screen "滑块角度" 800x480
   Circle "圆_2" at 245,51 size 21x21
      Appearance <- "360"
   Circle "圆_3" at 274,56 size 21x21
      Appearance <- "10度"
   Circle "圆_4" at 303,66 size 21x21
      Appearance <- "20度"
   Circle "圆_5" at 326,79 size 21x21
      Appearance <- "30度"
   Circle "圆_6" at 346,95 size 21x21
      Appearance <- "40度"
   Circle "圆_7" at 364,115 size 21x21
      Appearance <- "50"
   Circle "圆_8" at 377,135 size 21x21
      Appearance <- "60"
   Circle "圆_9" at 385,157 size 21x21
      Appearance <- "70"
   Circle "圆_10" at 392,179 size 21x21
      Appearance <- "80"
   Circle "圆_11" at 394,202 size 21x21
      Appearance <- "90"
   Circle "圆_12" at 391,226 size 21x21
      Appearance <- "100"
   Circle "圆_13" at 386,249 size 21x21
      Appearance <- "110"
   Circle "圆_14" at 378,271 size 21x21
      Appearance <- "120"
   Circle "圆_15" at 365,292 size 21x21
      Appearance <- "130"
   Circle "圆_16" at 348,311 size 21x21
      Appearance <- "140"
   Circle "圆_17" at 328,328 size 21x21
      Appearance <- "150"
   Circle "圆_18" at 306,342 size 21x21
      Appearance <- "160"
   Circle "圆_19" at 276,353 size 21x21
      Appearance <- "170"
   Circle "圆_20" at 247,357 size 21x21
      Appearance <- "180"
   Circle "圆_22" at 219,352 size 21x21
      Appearance <- "190"
   Circle "圆_23" at 195,344 size 21x21
      Appearance <- "200"
   Circle "圆_24" at 172,333 size 21x21
      Appearance <- "210"
   Circle "圆_25" at 152,319 size 21x21
      Appearance <- "220"
   Circle "圆_26" at 133,302 size 21x21
      Appearance <- "230"
   Circle "圆_27" at 117,281 size 21x21
      Appearance <- "240"
   Circle "圆_28" at 104,258 size 21x21
      Appearance <- "250"
   Circle "圆_29" at 96,229 size 21x21
      Appearance <- "260"
   Circle "圆_30" at 93,201 size 21x21
      Appearance <- "270"
   Circle "圆_32" at 95,178 size 21x21
      Appearance <- "280"
   Circle "圆_33" at 100,155 size 21x21
      Appearance <- "290"
   Circle "圆_34" at 110,131 size 21x21
      Appearance <- "300"
   Circle "圆_35" at 126,111 size 21x21
      Appearance <- "310"
   Circle "圆_36" at 144,91 size 21x21
      Appearance <- "320"
   Circle "圆_37" at 167,74 size 21x21
      Appearance <- "330"
   Circle "圆_38" at 191,63 size 21x21
      Appearance <- "340"
   Circle "圆_39" at 218,54 size 21x21
      Appearance <- "350"
   TextField "文本域_2" at 422,193 size 43x40; Text '90'
   TextField "文本域_3" at 221,378 size 62x40; Text '180'
   TextField "文本域_5" at 196,174 size 117x31; Text '滑块位置'
   TextField "文本域_9" at 467,193 size 93x25; Text '当前产量'
   TextField "文本域_4" at 25,203 size 62x40; Text '270'
   TextField "文本域_1" at 241,12 size 24x40; Text '0'
   SymbolLibrary "符号库_1" at 405,7 size 109x71
   SymbolLibrary "符号库_2" at 646,29 size 86x40
   TextField "文本域_7" at 637,83 size 77x21; Text '滑块电机'
   TextField "文本域_6" at 423,85 size 59x21; Text '主电机'
   TextField "文本域_8" at 467,127 size 93x25; Text '设置产量'
   TextField "文本域_10" at 693,127 size 93x25; Text '计数清零'
   TextField "文本域_13" at 586,126 size 93x25; Text '计数通断'
   TextField "文本域_11" at 35,338 size 93x25; Text '润滑检测'
   TextField "文本域_12" at 454,341 size 85x23; Text '润滑故障'
   TextField "文本域_15" at 583,14 size 33x17; Text '向上'
   TextField "文本域_16" at 738,15 size 33x17; Text '向下'
   Button "按钮_1" at 28,424 size 67x56; TextOff '滑块角度'
      on Click: ActivateScreen("滑块角度", 0)
   Button "按钮_2" at 96,424 size 67x56; TextOff '设备状态'
      on Click: ActivateScreen("设备状态", 0)
   Button "按钮_3" at 163,424 size 71x55; TextOff '工作台操作'
      on Click: ActivateScreen("工作台操作", 0)
   Button "按钮_4" at 235,424 size 69x56; TextOff '气垫操作'
      on Click: ActivateScreen("气垫操作", 0)
   Button "按钮_5" at 304,423 size 66x57; TextOff '故障显示'
      on Click: ActivateScreen("故障显示", 0)
   Button "按钮_6" at 371,423 size 73x57; TextOff '输出显示'
      on Click: ActivateScreen("输出显示", 0)
   Button "按钮_7" at 445,422 size 66x58; TextOff '输入显示'
      on Click: ActivateScreen("输入显示", 0)
   IOField "I/O 域_1" at 228,215 size 56x32; FormatPattern 999
      ProcessValue <- "横梁编码器 _DB_0.11"
   IOField "I/O 域_2" at 478,153 size 81x29; FormatPattern 9999
      ProcessValue <- "ECamdata _DB_设置产量"
   Button "按钮_8" at 514,423 size 68x56; TextOn '滑块调整'; TextOff '滑块调整'
      on Click: ActivateScreen("滑块调整", 0)
   Button "按钮_9" at 667,421 size 65x58; TextOff '报警信息'
      on Click: ActivateScreen("报警信息", 0)
   Button "按钮_10" at 585,423 size 77x55; TextOff '行程控制'
      on Click: ActivateScreen("行程控制", 0)
   Circle "圆_1" at 436,26 size 35x35
      Appearance <- "主电机正转运行"
   Circle "圆_21" at 584,33 size 33x33
      Appearance <- "滑块调整向上"
   Circle "圆_31" at 738,34 size 33x33
      Appearance <- "滑块调整向下"
   IOField "I/O 域_3" at 478,219 size 87x32; FormatPattern 9999
      ProcessValue <- "IEC_Counter_0_DB_4_CV"
   Rectangle "矩形_1" at 479,258 size 88x60
      Appearance <- "产量到达"
   TextField "文本域_14" at 478,277 size 85x23; Text '产量完成'
   Switch "开关_1" at 579,170 size 102x93; CaptionText 'Switch'; TextOff '断'; TextOn '通'
      ProcessValue <- "计数开始"
      Appearance <- "计数开始"
   Button "按钮_11" at 702,187 size 75x72; TextOff '清零'
      on Press: SetBit("计数清零")
      on Release: ResetBit("计数清零")
   Circle "圆_42" at 23,374 size 35x35
      Appearance <- "横梁1分油器检测"
   Circle "圆_43" at 129,375 size 35x35
      Appearance <- "平衡器分油器检测"
   Circle "圆_44" at 481,373 size 35x35
      Appearance <- "润滑正常"
   Circle "圆_45" at 230,100 size 55x55
      Appearance <- "上死点"
   TextField "文本域_17" at 233,118 size 47x17; Text '上死点'
   Circle "圆_46" at 229,274 size 55x55
      Appearance <- "下死点"
   TextField "文本域_18" at 232,292 size 47x17; Text '下死点'
   TextField "文本域_19" at 621,339 size 85x23; Text '平衡气压'
   Circle "圆_47" at 657,374 size 35x35
      Appearance <- "平衡缸气压检测"
   TextField "文本域_20" at 705,339 size 85x23; Text '液压保护'
   Circle "圆_48" at 737,373 size 35x35
      Appearance <- "液压保护故障(1)"
   TextField "文本域_21" at 539,340 size 85x23; Text '离制压力'
   Circle "圆_49" at 568,372 size 35x35
      Appearance <- "离制压力正常"
   TextField "文本域_22" at 370,342 size 85x23; Text '急停故障'
   Circle "圆_50" at 405,372 size 35x35
      Appearance <- "安全正常(1)"
   Circle "圆_51" at 78,375 size 35x35
      Appearance <- "滑块分油器检测"
   TextField "文本域_23" at 24,385 size 33x17; Text '横梁'
   TextField "文本域_24" at 78,385 size 33x17; Text '滑块'
   TextField "文本域_25" at 124,385 size 47x17; Text '平衡缸'
   Button "按钮_12" at 740,434 size 56x44; TextOff '润滑状态'
      on Click: ActivateScreen("润滑状态", 0)

screen "设备状态" 800x480
   TextField "文本域_1" at 63,79 size 101x27; Text '润滑正常'
   TextField "文本域_2" at 64,142 size 101x27; Text '急停正常'
   TextField "文本域_3" at 50,205 size 125x27; Text '工作台夹紧'
   TextField "文本域_4" at 66,268 size 101x27; Text '气压正常'
   TextField "文本域_5" at 46,331 size 149x27; Text '液压保护正常'
   Circle "圆_1" at 325,208 size 27x27
      Appearance <- "工作台落到位前"
   TextField "文本域_6" at 293,237 size 96x16; Text '工作台前落到为'
   Circle "圆_2" at 427,207 size 27x27
      Appearance <- "工作台落到位后"
   TextField "文本域_7" at 395,237 size 96x16; Text '工作台后落到为'
   TextField "文本域_8" at 495,237 size 96x16; Text '工作台夹紧压力'
   Circle "圆_4" at 223,207 size 27x27
      Appearance <- "工作台夹紧阀(1)"
   TextField "文本域_9" at 198,237 size 83x16; Text '工作台夹紧阀'
   Circle "圆_5" at 427,81 size 27x27
      Appearance <- "润滑油压正常"
   TextField "文本域_10" at 399,111 size 83x16; Text '润滑油压正常'
   TextField "文本域_12" at 295,111 size 96x16; Text '润滑过滤器正常'
   Circle "圆_8" at 222,81 size 27x27
      Appearance <- "工作台落到位后"
   TextField "文本域_13" at 196,111 size 83x16; Text '润滑油位正常'
   Circle "圆_9" at 527,81 size 27x27
      Appearance <- "工作台落到位后"
   TextField "文本域_14" at 502,111 size 83x16; Text '润滑频次正常'
   Circle "圆_10" at 325,270 size 27x27
      Appearance <- "工作台落到位前"
   TextField "文本域_15" at 306,299 size 70x16; Text '离合器压力'
   Circle "圆_11" at 427,269 size 27x27
      Appearance <- "工作台落到位后"
   Circle "圆_12" at 223,269 size 27x27
      Appearance <- "平衡缸气压检测"
   TextField "文本域_16" at 200,298 size 70x16; Text '平衡缸压力'
   TextField "文本域_17" at 407,300 size 70x16; Text '制动器压力'
   Circle "圆_6" at 615,81 size 27x27
      Appearance <- "润滑油泵启动OK"
   TextField "文本域_11" at 590,111 size 83x16; Text '润滑电机启动'
   TextField "文本域_19" at 312,171 size 57x16; Text '急停闭点'
   TextField "文本域_20" at 207,171 size 57x16; Text '急停开点'
   TextField "文本域_21" at 414,171 size 57x16; Text '梯子开关'
   TextField "文本域_23" at 306,362 size 70x16; Text '卸荷阀卸荷'
   Circle "圆_19" at 427,332 size 27x27
      Appearance <- "液压保护故障"
   TextField "文本域_24" at 200,361 size 83x16; Text '液压保护压力'
   TextField "文本域_25" at 407,363 size 57x16; Text '系统压力'
   Button "按钮_1" at 28,424 size 67x56; TextOn '滑块角度'; TextOff '滑块角度'
      on Click: ActivateScreen("滑块角度", 0)
   Button "按钮_2" at 96,424 size 67x56; TextOn '设备状态'; TextOff '设备状态'
      on Click: ActivateScreen("设备状态", 0)
   Button "按钮_3" at 163,424 size 71x55; TextOn '工作台操作'; TextOff '工作台操作'
      on Click: ActivateScreen("工作台操作", 0)
   Button "按钮_4" at 235,424 size 69x56; TextOn '气垫操作'; TextOff '气垫操作'
      on Click: ActivateScreen("气垫操作", 0)
   Button "按钮_5" at 304,423 size 66x57; TextOn '故障显示'; TextOff '故障显示'
      on Click: ActivateScreen("故障显示", 0)
   Button "按钮_6" at 371,423 size 73x57; TextOn '输出显示'; TextOff '输出显示'
      on Click: ActivateScreen("输出显示", 0)
   Button "按钮_7" at 445,422 size 66x58; TextOn '输入显示'; TextOff '输入显示'
      on Click: ActivateScreen("输入显示", 0)
   Button "按钮_8" at 514,423 size 68x56; TextOn '滑块调整'; TextOff '滑块调整'
      on Click: ActivateScreen("滑块调整", 0)
   Button "按钮_9" at 592,422 size 65x58; TextOn '报警信息'; TextOff '报警信息'
      on Click: ActivateScreen("报警信息", 0)

screen "输入显示" 800x480
   Button "按钮_1" at 28,424 size 67x56; TextOn '滑块角度'; TextOff '滑块角度'
      on Click: ActivateScreen("滑块角度", 0)
   Button "按钮_2" at 96,424 size 67x56; TextOn '设备状态'; TextOff '设备状态'
      on Click: ActivateScreen("设备状态", 0)
   Button "按钮_3" at 163,424 size 71x55; TextOn '工作台操作'; TextOff '工作台操作'
      on Click: ActivateScreen("工作台操作", 0)
   Button "按钮_4" at 235,424 size 69x56; TextOn '气垫操作'; TextOff '气垫操作'
      on Click: ActivateScreen("气垫操作", 0)
   Button "按钮_5" at 304,423 size 66x57; TextOn '故障显示'; TextOff '故障显示'
      on Click: ActivateScreen("故障显示", 0)
   Button "按钮_6" at 371,423 size 73x57; TextOn '输出显示'; TextOff '输出显示'
      on Click: ActivateScreen("输出显示", 0)
   Button "按钮_7" at 445,422 size 66x58; TextOn '输入显示'; TextOff '输入显示'
      on Click: ActivateScreen("输入显示", 0)
   Button "按钮_8" at 514,423 size 68x56; TextOn '滑块调整'; TextOff '滑块调整'
      on Click: ActivateScreen("滑块调整", 0)
   Button "按钮_9" at 592,422 size 65x58; TextOn '报警信息'; TextOff '报警信息'
      on Click: ActivateScreen("报警信息", 0)
   TextField "文本域_1" at 10,10 size 112x19; Text '主电机零速'
      Appearance <- "主电机零速"
   TextField "文本域_2" at 10,40 size 117x19; Text '主电机温度检测'
      Appearance <- "主电机温度检测(1)"
   TextField "文本域_3" at 10,70 size 117x19; Text '调速装置正常'
      Appearance <- "主电机调速装置正常"
   TextField "文本域_4" at 10,100 size 117x19; Text '主电机风扇空开'
      Appearance <- "主电机风扇空开"
   TextField "文本域_5" at 10,130 size 117x19; Text '风扇流量检测'
      Appearance <- "主电机风扇流量检测(1)"
   TextField "文本域_8" at 10,220 size 112x19; Text '按钮站插入'
      Appearance <- "按钮站插入"
   TextField "文本域_9" at 10,250 size 112x19; Text '右前急停按钮'
      Appearance <- "右前急停按钮"
   TextField "文本域_10" at 10,280 size 112x19; Text '左前急停按钮'
      Appearance <- "左前急停按钮"
   TextField "文本域_11" at 10,310 size 112x19; Text '右后急停按钮'
      Appearance <- "右后急停按钮"
   TextField "文本域_12" at 10,340 size 112x19; Text '左后急停按钮'
      Appearance <- "左后急停按钮"
   TextField "文本域_13" at 10,370 size 112x19; Text '前安全栓'
      Appearance <- "前安全栓"
   TextField "文本域_14" at 10,400 size 112x19; Text '后安全栓'
      Appearance <- "后安全栓"
   TextField "文本域_15" at 150,220 size 119x19; Text '气垫调整空开'
      Appearance <- "气垫调整空开"
   TextField "文本域_16" at 150,250 size 119x19; Text '气垫调整上极限'
      Appearance <- "气垫调整上极限"
   TextField "文本域_17" at 150,280 size 119x19; Text '气垫调整上极限'
      Appearance <- "气垫调整下极限"
   TextField "文本域_18" at 150,310 size 119x19; Text '冷却电机过热'
      Appearance <- "气垫冷却电机过热"
   TextField "文本域_19" at 150,340 size 119x19; Text '气垫左落下到位'
      Appearance <- "气垫左落下到位"
   TextField "文本域_20" at 150,370 size 119x19; Text '气垫左落下到位'
      Appearance <- "气垫左落下到位"
   TextField "文本域_21" at 150,400 size 119x19; Text '气垫压力检测'
      Appearance <- "气垫压力检测"
   TextField "文本域_22" at 290,220 size 117x19; Text '工作台开进到位'
      Appearance <- "工作台开进到位"
   TextField "文本域_23" at 290,250 size 117x19; Text '左前落到为'
      Appearance <- "工作台左前落到为"
   TextField "文本域_24" at 290,280 size 117x19; Text '右前落到为'
      Appearance <- "工作台右前落到为"
   TextField "文本域_25" at 290,310 size 117x19; Text '左后落到为'
      Appearance <- "工作台左后落到为"
   TextField "文本域_26" at 290,340 size 117x19; Text '右后落到位'
      Appearance <- "工作台右后落到位"
   TextField "文本域_27" at 290,370 size 117x19; Text '工作台落下夹紧'
      Appearance <- "工作台落下夹紧(1)"
   TextField "文本域_29" at 430,220 size 114x19; Text '液保空开'
      Appearance <- "液压保护系统空开"
   TextField "文本域_30" at 430,250 size 114x19; Text '50/AR液保压力'
      Appearance <- "50/AR液压保护压力"
   TextField "文本域_31" at 430,280 size 114x19; Text '90/AR液保压力'
      Appearance <- "90/AR液压保护压力"
   TextField "文本域_32" at 430,310 size 123x19; Text '100/AR液保压力'
      Appearance <- "100/AR液压保护压力"
   TextField "文本域_33" at 430,340 size 123x19; Text '135/AR液保压力'
      Appearance <- "135/AR液压保护压力"
   TextField "文本域_34" at 430,370 size 123x19; Text '150/AR液保压力'
      Appearance <- "150/AR液压保护压力"
   TextField "文本域_35" at 430,400 size 117x19; Text '平衡缸气压检测'
      Appearance <- "平衡缸气压检测"
   TextField "文本域_37" at 570,250 size 117x19; Text '离合器运行'
      Appearance <- "离合器运行"
   TextField "文本域_38" at 570,280 size 117x19; Text '离合器准确检测'
      Appearance <- "离合器准确检测"
   TextField "文本域_39" at 570,310 size 117x19; Text '离合冷却过滤器'
      Appearance <- "离合冷却过滤器检测"
   TextField "文本域_43" at 150,10 size 119x19; Text '滑块调整空开'
      Appearance <- "滑块调整电机空开"
   TextField "文本域_44" at 150,40 size 119x19; Text '滑块调整选择'
      Appearance <- "滑块调整选择开关"
   TextField "文本域_45" at 150,70 size 119x19; Text '滑块调整向上'
      Appearance <- "滑块调整向上"
   TextField "文本域_46" at 150,100 size 119x19; Text '滑块调整向下'
      Appearance <- "滑块调整向下"
   TextField "文本域_47" at 150,130 size 119x19; Text '滑块调整上极限'
      Appearance <- "滑块调整上极限"
   TextField "文本域_48" at 150,160 size 119x19; Text '滑块调整下极限'
      Appearance <- "滑块调整下极限"
   TextField "文本域_50" at 290,10 size 115x19; Text '工作台顶起压力'
      Appearance <- "工作台顶起压力"
   TextField "文本域_51" at 290,40 size 115x19; Text '左前顶起到位'
      Appearance <- "工作台左前顶起到位"
   TextField "文本域_52" at 290,70 size 115x19; Text '右前顶起到位'
      Appearance <- "工作台右前顶起到位"
   TextField "文本域_53" at 290,100 size 115x19; Text '左后顶起到位'
      Appearance <- "工作台左后顶起到位"
   TextField "文本域_54" at 290,130 size 115x19; Text '右后顶起到位'
      Appearance <- "工作台右后顶起到位"
   TextField "文本域_57" at 430,10 size 101x19; Text '润滑电机空开'
      Appearance <- "润滑电机空开"
   TextField "文本域_58" at 430,40 size 101x19; Text '润滑油位检测'
      Appearance <- "润滑油位检测"
   TextField "文本域_59" at 430,70 size 101x19; Text '润滑过滤检测'
      Appearance <- "润滑过滤检测"
   TextField "文本域_60" at 430,100 size 101x19; Text '滑块分油器'
      Appearance <- "滑块分油器检测"
   TextField "文本域_61" at 430,130 size 101x19; Text '平衡器分油器'
      Appearance <- "平衡器分油器检测"
   TextField "文本域_62" at 430,160 size 101x19; Text '气垫分油器'
      Appearance <- "气垫分油器检测"
   TextField "文本域_63" at 430,190 size 101x19; Text '横梁1分油器'
      Appearance <- "横梁1分油器检测"
   TextField "文本域_64" at 570,10 size 117x19; Text '离制压力检测'
      Appearance <- "离制压力检测"
   TextField "文本域_65" at 570,40 size 117x19; Text '离制油位检测'
      Appearance <- "离制油箱油位检测"
   TextField "文本域_66" at 570,70 size 117x19; Text '离制油温检测'
      Appearance <- "离制油箱油温检测"
   TextField "文本域_67" at 570,100 size 117x19; Text '离制过滤器检测'
      Appearance <- "离制过滤器检测"
   TextField "文本域_68" at 570,130 size 117x19; Text '离制双阀反馈1'
      Appearance <- "离制双阀反馈1"
   TextField "文本域_69" at 570,160 size 117x19; Text '离制双阀反馈2'
      Appearance <- "离制双阀反馈2"
   TextField "文本域_70" at 569,220 size 117x19; Text '离合器油泵空开'
      Appearance <- "离合器油泵空开"
   TextField "文本域_6" at 290,160 size 115x19; Text '变频器正常'
      Appearance <- "开工作台变频器正常"

screen "输出显示" 800x480
   Button "按钮_1" at 28,424 size 67x56; TextOn '滑块角度'; TextOff '滑块角度'
      on Click: ActivateScreen("滑块角度", 0)
   Button "按钮_2" at 96,424 size 67x56; TextOn '设备状态'; TextOff '设备状态'
      on Click: ActivateScreen("设备状态", 0)
   Button "按钮_3" at 163,424 size 71x55; TextOn '工作台操作'; TextOff '工作台操作'
      on Click: ActivateScreen("工作台操作", 0)
   Button "按钮_4" at 235,424 size 69x56; TextOn '气垫操作'; TextOff '气垫操作'
      on Click: ActivateScreen("气垫操作", 0)
   Button "按钮_5" at 304,423 size 66x57; TextOn '故障显示'; TextOff '故障显示'
      on Click: ActivateScreen("故障显示", 0)
   Button "按钮_6" at 371,423 size 73x57; TextOn '输出显示'; TextOff '输出显示'
      on Click: ActivateScreen("输出显示", 0)
   Button "按钮_7" at 445,422 size 66x58; TextOn '输入显示'; TextOff '输入显示'
      on Click: ActivateScreen("输入显示", 0)
   Button "按钮_8" at 514,423 size 68x56; TextOn '滑块调整'; TextOff '滑块调整'
      on Click: ActivateScreen("滑块调整", 0)
   Button "按钮_9" at 592,422 size 65x58; TextOn '报警信息'; TextOff '报警信息'
      on Click: ActivateScreen("报警信息", 0)
   TextField "文本域_1" at 10,10 size 101x19; Text '平衡缸进气阀'
      Appearance <- "平衡缸进气阀"
   TextField "文本域_2" at 10,40 size 101x19; Text '平衡缸排气阀'
      Appearance <- "平衡缸排气阀"
   TextField "文本域_3" at 10,70 size 101x19; Text '左气垫进气阀'
      Appearance <- "左气垫进气阀"
   TextField "文本域_4" at 10,100 size 101x19; Text '左气垫排气阀'
      Appearance <- "左气垫排气阀"
   TextField "文本域_5" at 10,130 size 101x19; Text '右气垫进气阀'
      Appearance <- "右气垫进气阀"
   TextField "文本域_6" at 11,156 size 101x19; Text '右气垫排气阀'
      Appearance <- "右气垫气排阀"
   TextField "文本域_7" at 12,218 size 101x19; Text '气动泵气源阀'
      Appearance <- "气动泵气源阀-1#"
   TextField "文本域_8" at 12,248 size 117x19; Text '液保启动卸荷阀'
      Appearance <- "液压保护泵启动（卸载）阀-2#"
   TextField "文本域_9" at 12,278 size 85x19; Text '液保负荷阀'
      Appearance <- "液压保护负荷荷 阀-3#"
   TextField "文本域_10" at 12,308 size 117x19; Text '工作台放松顶起'
      Appearance <- "工作台放松顶起(1)"
   TextField "文本域_11" at 12,338 size 117x19; Text '工作台落下夹紧'
      Appearance <- "工作台落下夹紧(1)"
   TextField "文本域_12" at 13,364 size 85x19; Text '工作台顶起'
      Appearance <- "工作台顶起"
   TextField "文本域_13" at 14,391 size 85x19; Text '工作台落下'
      Appearance <- "工作台落下夹紧(2)"
   TextField "文本域_14" at 152,10 size 117x19; Text '气垫间歇润滑阀'
      Appearance <- "气垫间歇润滑阀"
   TextField "文本域_15" at 152,40 size 85x19; Text '自动化气压'
      Appearance <- "自动化气压"
   TextField "文本域_16" at 152,70 size 117x19; Text '主电机启动指示'
      Appearance <- "主电机启动指示"
   TextField "文本域_17" at 152,100 size 101x19; Text '飞轮停止指示'
      Appearance <- "飞轮停止指示灯"
   TextField "文本域_18" at 152,130 size 101x19; Text '模具移出指示'
      Appearance <- "模具移出指示"
   TextField "文本域_19" at 153,156 size 101x19; Text '模具装入指示'
      Appearance <- "模具装入指示"
   TextField "文本域_20" at 149,183 size 133x19; Text '润滑电机工作指示'
      Appearance <- "润滑电机工作指示"
   TextField "文本域_21" at 10,183 size 133x19; Text '平衡缸间歇润滑阀'
      Appearance <- "平衡器间歇润滑阀"
   TextField "文本域_22" at 157,219 size 133x19; Text '液压保护正常指示'
      Appearance <- "液压保护正常指示"
   TextField "文本域_23" at 157,249 size 133x19; Text '液压保护卸荷指示'
      Appearance <- "液压保护卸荷指示"
   TextField "文本域_24" at 157,279 size 85x19; Text '气垫升指示'
      Appearance <- "气垫升"
   TextField "文本域_25" at 157,309 size 85x19; Text '气垫降指示'
      Appearance <- "气垫降"
   TextField "文本域_26" at 157,339 size 85x19; Text '飞轮制动阀'
      Appearance <- "飞轮制动阀"
   TextField "文本域_27" at 158,365 size 69x19; Text '单人操作'
      Appearance <- "单人操作"
   TextField "文本域_28" at 154,392 size 85x19; Text '气垫电机升'
      Appearance <- "气垫升(1)"
   TextField "文本域_29" at 297,12 size 85x19; Text '气垫电机降'
      Appearance <- "气垫降(1)"
   TextField "文本域_30" at 297,42 size 85x19; Text '主电机运行'
      Appearance <- "主电机正转运行"
   TextField "文本域_31" at 297,72 size 69x19; Text '速度控制'
      Appearance <- "速度控制"
   TextField "文本域_32" at 297,102 size 85x19; Text '主电机反转'
      Appearance <- "主电机反转"
   TextField "文本域_33" at 297,132 size 85x19; Text '主电机正转'
      Appearance <- "主电机正转运行"
   TextField "文本域_34" at 298,158 size 85x19; Text '系统泵开始'
      Appearance <- "系统泵开始"
   TextField "文本域_35" at 294,185 size 101x19; Text '工台变频使能'
      Appearance <- "变频器使能"
   TextField "文本域_36" at 299,222 size 101x19; Text '工台电机正转'
      Appearance <- "工作台电机正转(1)"
   TextField "文本域_37" at 299,252 size 101x19; Text '工台电机反转'
      Appearance <- "工作骀电机反转"
   TextField "文本域_38" at 299,282 size 85x19; Text '工作台变速'
      Appearance <- "工作台变速"
   TextField "文本域_39" at 299,312 size 101x19; Text '润滑电机运行'
      Appearance <- "润滑电机"
   TextField "文本域_40" at 299,342 size 69x19; Text '安全正常'
      Appearance <- "安全正常(1)"
   TextField "文本域_41" at 300,368 size 78x19; Text '压机急停1'
      Appearance <- "压机急停1"
   TextField "文本域_42" at 296,395 size 78x19; Text '压机急停2'
      Appearance <- "压机急停2"
   TextField "文本域_43" at 439,13 size 117x19; Text '离合器油泵电机'
      Appearance <- "离合器油泵电机"
   TextField "文本域_44" at 439,43 size 117x19; Text '单次连续继电器'
      Appearance <- "单次连续继电器"
   TextField "文本域_45" at 439,73 size 101x19; Text '滑块向上调整'
      Appearance <- "滑块向上调整"
   TextField "文本域_46" at 439,103 size 101x19; Text '滑块向下调整'
      Appearance <- "滑块向下调整"
   TextField "文本域_47" at 439,133 size 117x19; Text '主电机风扇运行'
      Appearance <- "主电机风扇运行"

screen "故障显示" 800x480
   Button "按钮_1" at 28,424 size 67x56; TextOn '滑块角度'; TextOff '滑块角度'
      on Click: ActivateScreen("滑块角度", 0)
   Button "按钮_2" at 96,424 size 67x56; TextOn '设备状态'; TextOff '设备状态'
      on Click: ActivateScreen("设备状态", 0)
   Button "按钮_3" at 163,424 size 71x55; TextOn '工作台操作'; TextOff '工作台操作'
      on Click: ActivateScreen("工作台操作", 0)
   Button "按钮_4" at 235,424 size 69x56; TextOn '气垫操作'; TextOff '气垫操作'
      on Click: ActivateScreen("气垫操作", 0)
   Button "按钮_5" at 304,423 size 66x57; TextOn '故障显示'; TextOff '故障显示'
      on Click: ActivateScreen("故障显示", 0)
   Button "按钮_6" at 371,423 size 73x57; TextOn '输出显示'; TextOff '输出显示'
      on Click: ActivateScreen("输出显示", 0)
   Button "按钮_7" at 445,422 size 66x58; TextOn '输入显示'; TextOff '输入显示'
      on Click: ActivateScreen("输入显示", 0)
   Button "按钮_8" at 514,423 size 68x56; TextOn '滑块调整'; TextOff '滑块调整'
      on Click: ActivateScreen("滑块调整", 0)
   Button "按钮_9" at 592,422 size 65x58; TextOn '报警信息'; TextOff '报警信息'
      on Click: ActivateScreen("报警信息", 0)

screen "工作台操作" 800x480
   Button "按钮_1" at 28,424 size 67x56; TextOn '滑块角度'; TextOff '滑块角度'
      on Click: ActivateScreen("滑块角度", 0)
   Button "按钮_2" at 96,424 size 67x56; TextOn '设备状态'; TextOff '设备状态'
      on Click: ActivateScreen("设备状态", 0)
   Button "按钮_3" at 163,424 size 71x55; TextOn '工作台操作'; TextOff '工作台操作'
      on Click: ActivateScreen("工作台操作", 0)
   Button "按钮_4" at 235,424 size 69x56; TextOn '气垫操作'; TextOff '气垫操作'
      on Click: ActivateScreen("气垫操作", 0)
   Button "按钮_5" at 304,423 size 66x57; TextOn '故障显示'; TextOff '故障显示'
      on Click: ActivateScreen("故障显示", 0)
   Button "按钮_6" at 371,423 size 73x57; TextOn '输出显示'; TextOff '输出显示'
      on Click: ActivateScreen("输出显示", 0)
   Button "按钮_7" at 445,422 size 66x58; TextOn '输入显示'; TextOff '输入显示'
      on Click: ActivateScreen("输入显示", 0)
   TextField "文本域_1" at 47,68 size 125x27; Text '工作台松开'
   TextField "文本域_2" at 53,142 size 125x27; Text '工作台夹紧'
   Circle "圆_7" at 315,60 size 27x27
      Appearance <- "工作台放松顶起"
   TextField "文本域_12" at 308,92 size 44x16; Text '工作台'
   Circle "圆_8" at 222,60 size 27x27
      Appearance <- "上死点"
   TextField "文本域_13" at 215,92 size 44x16; Text '上死点'
   TextField "文本域_14" at 576,92 size 44x16; Text '工作台'
   Circle "圆_6" at 635,60 size 27x27
      Appearance <- "工作台放松OK"
   TextField "文本域_11" at 628,92 size 44x16; Text '工作台'
   Button "按钮_8" at 514,423 size 68x56; TextOn '滑块调整'; TextOff '滑块调整'
      on Click: ActivateScreen("滑块调整", 0)
   Button "按钮_9" at 592,422 size 65x58; TextOn '报警信息'; TextOff '报警信息'
      on Click: ActivateScreen("报警信息", 0)
   Circle "圆_1" at 271,60 size 27x27
      Appearance <- "调整开关"
   TextField "文本域_5" at 268,93 size 31x16; Text '调整'
   Circle "圆_3" at 582,60 size 27x27
      Appearance <- "工作台顶起压力"
   TextField "文本域_6" at 267,110 size 33x17; Text '开关'
   TextField "文本域_7" at 312,109 size 33x17; Text '顶起'
   TextField "文本域_8" at 574,110 size 47x17; Text '松压力'
   TextField "文本域_10" at 397,91 size 31x16; Text '前左'
   Circle "圆_4" at 399,60 size 27x27
      Appearance <- "工作台左前顶起到位"
   TextField "文本域_15" at 392,108 size 47x17; Text '松到位'
   TextField "文本域_16" at 443,91 size 31x16; Text '前右'
   Circle "圆_5" at 443,60 size 27x27
      Appearance <- "工作台右前顶起到位"
   TextField "文本域_17" at 438,109 size 47x17; Text '松到位'
   TextField "文本域_18" at 488,91 size 31x16; Text '后左'
   Circle "圆_9" at 489,60 size 27x27
      Appearance <- "工作台左后顶起到位"
   TextField "文本域_22" at 484,109 size 47x17; Text '松到位'
   TextField "文本域_23" at 535,91 size 31x16; Text '后右'
   Circle "圆_10" at 535,60 size 27x27
      Appearance <- "工作台右后顶起到位"
   TextField "文本域_24" at 530,109 size 47x17; Text '松到位'
   TextField "文本域_9" at 628,109 size 45x16; Text '松开OK'
   TextField "文本域_3" at 351,92 size 44x16; Text '工作台'
   Circle "圆_2" at 358,60 size 27x27
      Appearance <- "工作台放松顶起(1)"
   TextField "文本域_4" at 349,108 size 47x17; Text '松开阀'
   Circle "圆_11" at 268,141 size 27x27
      Appearance <- "工作台落下夹紧(1)"
   TextField "文本域_19" at 261,171 size 44x16; Text '工作台'
   TextField "文本域_21" at 529,170 size 44x16; Text '工作台'
   Circle "圆_13" at 588,141 size 27x27
      Appearance <- "工作台-夹紧OK"
   TextField "文本域_25" at 581,170 size 44x16; Text '工作台'
   Circle "圆_14" at 224,141 size 27x27
      Appearance <- "调整开关"
   TextField "文本域_26" at 217,171 size 44x16; Text '工作台'
   Circle "圆_15" at 535,141 size 27x27
      Appearance <- "工作台顶起压力"
   TextField "文本域_27" at 218,187 size 47x17; Text '进到位'
   TextField "文本域_28" at 265,187 size 33x17; Text '夹紧'
   TextField "文本域_29" at 527,188 size 47x17; Text '夹压力'
   TextField "文本域_30" at 350,171 size 31x16; Text '前左'
   Circle "圆_16" at 352,142 size 27x27
      Appearance <- "工作台落下左前检测"
   TextField "文本域_31" at 345,187 size 47x17; Text '落到位'
   TextField "文本域_32" at 396,171 size 31x16; Text '前右'
   Circle "圆_17" at 396,141 size 27x27
      Appearance <- "工作台落下右前检测"
   TextField "文本域_33" at 391,187 size 47x17; Text '落到位'
   TextField "文本域_34" at 441,170 size 31x16; Text '后左'
   Circle "圆_18" at 442,141 size 27x27
      Appearance <- "工作台落下左后检测"
   TextField "文本域_35" at 437,187 size 47x17; Text '落到位'
   TextField "文本域_36" at 488,170 size 31x16; Text '后右'
   Circle "圆_19" at 488,141 size 27x27
      Appearance <- "工作台落下右边后检测"
   TextField "文本域_37" at 483,188 size 47x17; Text '落到位'
   TextField "文本域_38" at 581,187 size 45x16; Text '夹紧OK'
   TextField "文本域_39" at 304,171 size 44x16; Text '工作台'
   Circle "圆_20" at 311,143 size 27x27
      Appearance <- "工作台落下夹紧(2)"
   TextField "文本域_40" at 302,187 size 47x17; Text '夹紧阀'
   TextField "文本域_20" at 52,232 size 125x27; Text '工作台开进'
   TextField "文本域_41" at 58,306 size 125x27; Text '工作台开出'
   Circle "圆_21" at 227,224 size 27x27
      Appearance <- "上死点"
   TextField "文本域_43" at 220,256 size 44x16; Text '上死点'
   Circle "圆_23" at 276,224 size 27x27
      Appearance <- "调整开关"
   TextField "文本域_46" at 273,257 size 31x16; Text '调整'
   TextField "文本域_47" at 272,274 size 33x17; Text '开关'
   TextField "文本域_50" at 402,255 size 44x16; Text '工作台'
   Circle "圆_25" at 404,224 size 27x27
      Appearance <- "工作台开进"
   TextField "文本域_51" at 397,272 size 35x17; Text '进'
   TextField "文本域_52" at 447,255 size 44x16; Text '工作台'
   Circle "圆_26" at 452,224 size 27x27
      Appearance <- "工作台开进到位"
   TextField "文本域_53" at 444,273 size 47x17; Text '进到位'
   TextField "文本域_59" at 356,256 size 44x16; Text '工台变'
   Circle "圆_29" at 363,224 size 27x27
      Appearance <- "开工作台变频器正常"
   TextField "文本域_60" at 354,272 size 47x17; Text '频正常'
   Circle "圆_12" at 316,224 size 27x27
      Appearance <- "工作台放松OK"
   TextField "文本域_42" at 309,256 size 44x16; Text '工作台'
   TextField "文本域_48" at 309,273 size 45x16; Text '松开OK'
   Circle "圆_22" at 230,305 size 27x27
      Appearance <- "上死点"
   TextField "文本域_44" at 223,337 size 44x16; Text '上死点'
   Circle "圆_24" at 279,305 size 27x27
      Appearance <- "调整开关"
   TextField "文本域_45" at 276,338 size 31x16; Text '调整'
   TextField "文本域_49" at 275,355 size 33x17; Text '开关'
   TextField "文本域_54" at 405,336 size 44x16; Text '工作台'
   Circle "圆_27" at 407,305 size 27x27
      Appearance <- "工作台开出"
   TextField "文本域_55" at 400,353 size 19x17; Text '出'
   TextField "文本域_56" at 450,336 size 44x16; Text '工作台'
   Circle "圆_28" at 455,305 size 27x27
      Appearance <- "工作台顶起右前检测"
   TextField "文本域_57" at 447,354 size 47x17; Text '出到位'
   TextField "文本域_58" at 359,337 size 44x16; Text '工台变'
   Circle "圆_30" at 366,305 size 27x27
      Appearance <- "开工作台变频器正常"
   TextField "文本域_61" at 357,353 size 47x17; Text '频正常'
   Circle "圆_31" at 319,305 size 27x27
      Appearance <- "工作台放松OK"
   TextField "文本域_62" at 312,337 size 44x16; Text '工作台'
   TextField "文本域_63" at 312,354 size 45x16; Text '松开OK'

screen "气垫操作" 800x480
   Button "按钮_1" at 28,424 size 67x56; TextOn '滑块角度'; TextOff '滑块角度'
      on Click: ActivateScreen("滑块角度", 0)
   Button "按钮_2" at 96,424 size 67x56; TextOn '设备状态'; TextOff '设备状态'
      on Click: ActivateScreen("设备状态", 0)
   Button "按钮_3" at 163,424 size 71x55; TextOn '工作台操作'; TextOff '工作台操作'
      on Click: ActivateScreen("工作台操作", 0)
   Button "按钮_4" at 235,424 size 69x56; TextOn '气垫操作'; TextOff '气垫操作'
      on Click: ActivateScreen("气垫操作", 0)
   Button "按钮_5" at 304,423 size 66x57; TextOn '故障显示'; TextOff '故障显示'
      on Click: ActivateScreen("故障显示", 0)
   Button "按钮_6" at 371,423 size 73x57; TextOn '输出显示'; TextOff '输出显示'
      on Click: ActivateScreen("输出显示", 0)
   Button "按钮_7" at 445,422 size 66x58; TextOn '输入显示'; TextOff '输入显示'
      on Click: ActivateScreen("输入显示", 0)
   Button "按钮_8" at 514,423 size 68x56; TextOn '滑块调整'; TextOff '滑块调整'
      on Click: ActivateScreen("滑块调整", 0)
   Button "按钮_9" at 592,422 size 65x58; TextOn '报警信息'; TextOff '报警信息'
      on Click: ActivateScreen("报警信息", 0)
   Ellipse "椭圆_1" at 16,71 size 119x42
      Appearance <- "气垫上调整"
   TextField "文本域_1" at 22,85 size 101x27; Text '气垫上调'
   Ellipse "椭圆_2" at 17,134 size 119x42
      Appearance <- "气垫下降调整"
   TextField "文本域_2" at 27,142 size 101x27; Text '气垫下调'
   TextField "文本域_13" at 209,111 size 44x16; Text '上死点'
   TextField "文本域_5" at 257,112 size 70x16; Text '气垫落到位'
   TextField "文本域_6" at 191,244 size 47x29; Text '190'
   TextField "文本域_9" at 11,244 size 161x29; Text '气垫调整上限'
   TextField "文本域_10" at 192,317 size 47x29; Text '380'
   TextField "文本域_11" at 13,317 size 161x29; Text '气垫调整下限'
   TextField "文本域_12" at 272,243 size 135x29; Text '气垫当前值'
   TextField "文本域_14" at 274,318 size 135x29; Text '气垫设定值'
   IOField "I/O 域_1" at 409,312 size 96x47; FormatPattern 9999
      ProcessValue <- "气垫编码器数据_气垫设定值"
   IOField "I/O 域_3" at 410,243 size 96x47; FormatPattern 9999
      ProcessValue <- "气垫编码器数据_气垫高度"
   Circle "圆_1" at 584,30 size 39x39
      Appearance <- "气垫调整自动"
   Circle "圆_2" at 690,31 size 39x39
      Appearance <- "气垫调整自动"
   TextField "文本域_16" at 583,76 size 41x21; Text '手动'
   TextField "文本域_19" at 689,76 size 41x21; Text '自动'
   Switch "开关_1" at 600,93 size 120x56; TextOn '自动'; CaptionText 'Switch'; TextOff '手动'
      on SwitchOff: ResetBit("滑块调整手动/自动")
      on SwitchOn: SetBit("滑块调整手动/自动")
      Appearance <- "滑块调整手动/自动"
      ProcessValue <- "气垫调整自动"
   TextField "文本域_7" at 599,150 size 123x21; Text '手动/自动调整'
   Circle "圆_4" at 214,68 size 37x37
      Appearance <- "上死点"
   Circle "圆_3" at 272,70 size 37x37
      Appearance <- "气垫左落下到位"
   TextField "文本域_8" at 328,112 size 83x16; Text '气垫调整空开'
   Circle "圆_5" at 342,70 size 37x37
      Appearance <- "气垫调整空开"
   TextField "文本域_15" at 411,112 size 57x16; Text '选择关闭'
   Circle "圆_6" at 420,71 size 37x37
      Appearance <- "选择关闭"
   TextField "文本域_17" at 467,112 size 70x16; Text '气垫上限位'
   Circle "圆_7" at 481,71 size 37x37
      Appearance <- "气垫调整上极限"
   TextField "文本域_3" at 209,179 size 44x16; Text '上死点'
   TextField "文本域_4" at 257,180 size 70x16; Text '气垫落到位'
   Circle "圆_8" at 214,136 size 37x37
      Appearance <- "上死点"
   Circle "圆_9" at 272,138 size 37x37
      Appearance <- "气垫左落下到位"
   TextField "文本域_18" at 328,180 size 83x16; Text '气垫调整空开'
   Circle "圆_10" at 342,138 size 37x37
      Appearance <- "气垫调整空开"
   TextField "文本域_20" at 411,180 size 57x16; Text '选择关闭'
   Circle "圆_11" at 420,139 size 37x37
      Appearance <- "选择关闭"
   TextField "文本域_21" at 467,180 size 70x16; Text '气垫下限位'
   Circle "圆_12" at 481,139 size 37x37
      Appearance <- "气垫调整下极限"
   TextField "文本域_22" at 150,110 size 57x16; Text '气垫选择'
   Circle "圆_13" at 155,70 size 37x37
      Appearance <- "气垫选择开关"
   TextField "文本域_23" at 150,178 size 57x16; Text '气垫选择'
   Circle "圆_14" at 155,138 size 37x37
      Appearance <- "气垫选择开关"

screen "滑块调整" 800x480
   Button "按钮_1" at 28,424 size 67x56; TextOn '滑块角度'; TextOff '滑块角度'
      on Click: ActivateScreen("滑块角度", 0)
   Button "按钮_2" at 96,424 size 67x56; TextOn '设备状态'; TextOff '设备状态'
      on Click: ActivateScreen("设备状态", 0)
   Button "按钮_3" at 163,424 size 71x55; TextOn '工作台操作'; TextOff '工作台操作'
      on Click: ActivateScreen("工作台操作", 0)
   Button "按钮_4" at 235,424 size 69x56; TextOn '气垫操作'; TextOff '气垫操作'
      on Click: ActivateScreen("气垫操作", 0)
   Button "按钮_5" at 304,423 size 66x57; TextOn '故障显示'; TextOff '故障显示'
      on Click: ActivateScreen("故障显示", 0)
   Button "按钮_6" at 371,423 size 73x57; TextOn '输出显示'; TextOff '输出显示'
      on Click: ActivateScreen("输出显示", 0)
   Button "按钮_7" at 445,422 size 66x58; TextOn '输入显示'; TextOff '输入显示'
      on Click: ActivateScreen("输入显示", 0)
   Button "按钮_8" at 514,423 size 68x56; TextOff '滑块调整'
      on Click: ActivateScreen("滑块调整", 0)
   TextField "文本域_1" at 157,34 size 61x29; Text '1220'
   TextField "文本域_2" at 26,34 size 109x29; Text '滑块上限'
   TextField "文本域_3" at 158,107 size 47x29; Text '560'
   TextField "文本域_4" at 27,107 size 109x29; Text '滑块下限'
   TextField "文本域_6" at 268,33 size 135x29; Text '滑块当前值'
   TextField "文本域_8" at 270,108 size 135x29; Text '滑块设定值'
   Circle "圆_1" at 584,30 size 39x39
      Appearance <- "滑块调整手动/自动"
   Circle "圆_2" at 690,31 size 39x39
      Appearance <- "滑块调整手动/自动"
   TextField "文本域_16" at 583,76 size 41x21; Text '手动'
   TextField "文本域_19" at 689,76 size 41x21; Text '自动'
   IOField "I/O 域_1" at 405,102 size 96x47; FormatPattern 9999
      ProcessValue <- "ECamdata _DB_D108"
   IOField "I/O 域_2" at 406,33 size 96x47; FormatPattern 9999
      ProcessValue <- "ECamdata _DB_D107"
   Switch "开关_1" at 600,93 size 120x56; CaptionText 'Switch'; TextOff '手动'; TextOn '自动'
      on SwitchOff: ResetBit("滑块调整手动/自动")
      on SwitchOn: SetBit("滑块调整手动/自动")
      Appearance <- "滑块调整手动/自动"
      ProcessValue <- "滑块调整手动/自动"
   TextField "文本域_5" at 599,150 size 123x21; Text '手动/自动调整'
   Button "按钮_10" at 592,422 size 65x58; TextOn '报警信息'; TextOff '报警信息'
      on Click: ActivateScreen("报警信息", 0)
   Circle "圆_3" at 32,276 size 33x33
      Appearance <- "平衡缸气压检测"
   TextField "文本域_7" at 8,8 size 37x17; Text 'Text'
   TextField "文本域_10" at 26,281 size 47x17; Text '平衡缸'
   Circle "圆_4" at 89,276 size 33x33
      Appearance <- "液压保护正常"
   TextField "文本域_11" at 80,281 size 47x17; Text '液压保'
   Circle "圆_5" at 143,276 size 33x33
      Appearance <- "润滑正常"
   TextField "文本域_12" at 144,280 size 33x17; Text '润滑'
   Circle "圆_6" at 199,276 size 33x33
      Appearance <- "滑块调整电机空开"
   TextField "文本域_13" at 197,283 size 33x17; Text '调整'
   Circle "圆_7" at 252,276 size 33x33
      Appearance <- "滑块调整选择开关"
   TextField "文本域_14" at 244,281 size 47x17; Text '滑块调'
   Circle "圆_8" at 303,263 size 33x33
      Appearance <- "上死点"
   TextField "文本域_15" at 295,269 size 47x17; Text '上死点'
   Circle "圆_9" at 407,265 size 33x33
      Appearance <- "滑块调整上极限"
   TextField "文本域_17" at 397,276 size 47x17; Text '上限位'
   Circle "圆_10" at 407,301 size 33x33
      Appearance <- "滑块调整下极限"
   TextField "文本域_18" at 396,315 size 47x17; Text '下限位'
   Circle "圆_11" at 496,260 size 33x33
      Appearance <- "滑块向上调整"
   TextField "文本域_20" at 485,271 size 61x17; Text '调整向上'
   Circle "圆_12" at 498,306 size 33x33
      Appearance <- "滑块向下调整"
   TextField "文本域_21" at 482,316 size 61x17; Text '调整向下'
   Circle "圆_13" at 354,277 size 33x33
      Appearance <- "急停故障"
   TextField "文本域_9" at 355,289 size 33x17; Text '急停'
   Circle "圆_14" at 448,245 size 37x37
      Appearance <- "滑块调整手动/自动"
   TextField "文本域_22" at 447,255 size 41x21; Text '手动'
   Circle "圆_15" at 448,283 size 37x37
      Appearance <- "滑块调整手动/自动"
   TextField "文本域_23" at 446,291 size 41x21; Text '自动'
   Circle "圆_16" at 448,322 size 38x38
      Appearance <- "滑块调整手动/自动"
   TextField "文本域_24" at 446,329 size 41x21; Text '手动'
   TextField "文本域_25" at 31,295 size 33x17; Text '气压'
   TextField "文本域_26" at 80,297 size 47x17; Text '护正常'
   TextField "文本域_27" at 144,296 size 33x17; Text '正常'
   TextField "文本域_28" at 198,297 size 33x17; Text '空开'
   TextField "文本域_29" at 246,297 size 47x17; Text '整选择'
   Circle "圆_17" at 302,300 size 33x33
      Appearance <- "下死点"
   TextField "文本域_30" at 294,306 size 47x17; Text '下死点'

screen "报警信息" 800x480
   AlarmView "报警视图_1" at 10,90 size 780x331
   Clock "时钟_1" at 630,64 size 164x20
   GraphicView "图形视图_2" at 2,9 size 78x46; Picture "方鼎LOGO"
   TextField "文本域_5" at 222,19 size 365x33; Text '湖北方鼎科技发展有限公司'
   TextField "文本域_3" at 710,9 size 75x21; Text 'SIEMENS'
   TextField "文本域_4" at 702,37 size 93x17; Text 'SIMATIC HMI'
   TextField "文本域_1" at 325,62 size 109x29; Text '报警信息'
   Button "按钮_1" at 28,424 size 67x56; TextOn '滑块角度'; TextOff '滑块角度'
      on Click: ActivateScreen("滑块角度", 0)
   Button "按钮_2" at 96,424 size 67x56; TextOn '设备状态'; TextOff '设备状态'
      on Click: ActivateScreen("设备状态", 0)
   Button "按钮_3" at 163,424 size 71x55; TextOn '工作台操作'; TextOff '工作台操作'
      on Click: ActivateScreen("工作台操作", 0)
   Button "按钮_4" at 235,424 size 69x56; TextOn '气垫操作'; TextOff '气垫操作'
      on Click: ActivateScreen("气垫操作", 0)
   Button "按钮_5" at 304,423 size 66x57; TextOn '故障显示'; TextOff '故障显示'
      on Click: ActivateScreen("故障显示", 0)
   Button "按钮_6" at 371,423 size 73x57; TextOn '输出显示'; TextOff '输出显示'
      on Click: ActivateScreen("输出显示", 0)
   Button "按钮_7" at 445,422 size 66x58; TextOn '输入显示'; TextOff '输入显示'
      on Click: ActivateScreen("输入显示", 0)
   Button "按钮_8" at 514,423 size 68x56; TextOn '滑块调整'; TextOff '滑块调整'
      on Click: ActivateScreen("滑块调整", 0)
   Button "按钮_9" at 592,422 size 65x58; TextOn '报警信息'; TextOff '报警信息'
      on Click: ActivateScreen("报警信息", 0)

screen "行程控制" 800x480
   Button "按钮_1" at 28,424 size 67x56; TextOn '滑块角度'; TextOff '滑块角度'
      on Click: ActivateScreen("滑块角度", 0)
   Button "按钮_2" at 96,424 size 67x56; TextOn '设备状态'; TextOff '设备状态'
      on Click: ActivateScreen("设备状态", 0)
   Button "按钮_3" at 163,424 size 71x55; TextOn '工作台操作'; TextOff '工作台操作'
      on Click: ActivateScreen("工作台操作", 0)
   Button "按钮_4" at 235,424 size 69x56; TextOn '气垫操作'; TextOff '气垫操作'
      on Click: ActivateScreen("气垫操作", 0)
   Button "按钮_5" at 304,423 size 66x57; TextOn '故障显示'; TextOff '故障显示'
      on Click: ActivateScreen("故障显示", 0)
   Button "按钮_6" at 371,423 size 73x57; TextOn '输出显示'; TextOff '输出显示'
      on Click: ActivateScreen("输出显示", 0)
   Button "按钮_7" at 445,422 size 66x58; TextOn '输入显示'; TextOff '输入显示'
      on Click: ActivateScreen("输入显示", 0)
   Button "按钮_8" at 514,423 size 68x56; TextOn '滑块调整'; TextOff '滑块调整'
      on Click: ActivateScreen("滑块调整", 0)
   Button "按钮_9" at 667,421 size 65x58; TextOn '报警信息'; TextOff '报警信息'
      on Click: ActivateScreen("报警信息", 0)
   Button "按钮_10" at 585,423 size 77x55; TextOn '行程控制'; TextOff '行程控制'
      on Click: ActivateScreen("行程控制", 0)
   Circle "圆_1" at 162,107 size 34x34
      Appearance <- "行程选择"
   TextField "文本域_1" at 153,147 size 61x17; Text '行程选择'
   Circle "圆_2" at 223,107 size 34x34
      Appearance <- "左后双手使用"
   TextField "文本域_2" at 214,147 size 61x17; Text '左前选择'
   Circle "圆_3" at 284,107 size 34x34
      Appearance <- "右前双手选择"
   TextField "文本域_3" at 275,147 size 61x17; Text '右前选择'
   Circle "圆_4" at 345,107 size 34x34
      Appearance <- "行程选择"
   TextField "文本域_4" at 336,147 size 61x17; Text '换模完成'
   Circle "圆_5" at 406,107 size 34x34
      Appearance <- "行程选择"
   TextField "文本域_5" at 397,147 size 61x17; Text '急停正常'
   Circle "圆_6" at 467,107 size 34x34
      Appearance <- "行程选择"
   TextField "文本域_6" at 453,163 size 75x17; Text '主电机运行'
   Circle "圆_7" at 528,107 size 34x34
      Appearance <- "行程选择"
   TextField "文本域_7" at 519,147 size 61x17; Text '设备正常'
   Circle "圆_8" at 589,107 size 34x34
      Appearance <- "行程选择"
   TextField "文本域_8" at 580,147 size 61x17; Text '润滑正常'
   Button "按钮_11" at 0,3 size 165x55; TextOn '行程控制'; TextOff '行程控制'
      on Click: ActivateScreen("行程控制", 0)
   TextField "文本域_20" at 318,71 size 125x27; Text '主电机启动'

screen "主电机启动" 800x480
   TextField "文本域_20" at 111,181 size 125x27; Text '主电机启动'
   Circle "圆_21" at 286,176 size 33x33
      Appearance <- "润滑正常"
   TextField "文本域_43" at 279,231 size 57x16; Text '润滑正常'
   Circle "圆_23" at 346,176 size 33x33
      Appearance <- "调整开关"
   TextField "文本域_46" at 343,232 size 44x16; Text '润滑正'
   TextField "文本域_47" at 342,249 size 47x17; Text '常指示'
   TextField "文本域_50" at 523,230 size 57x16; Text '启动延时'
   Circle "圆_25" at 525,175 size 35x35
      Appearance <- "工作台开进"
   TextField "文本域_52" at 584,230 size 70x16; Text '主电机运行'
   Circle "圆_26" at 589,175 size 35x35
      Appearance <- "工作台开进到位"
   TextField "文本域_59" at 456,231 size 57x16; Text '变频上电'
   Circle "圆_29" at 463,176 size 34x34
      Appearance <- "开工作台变频器正常"
   Circle "圆_12" at 404,176 size 33x33
      Appearance <- "工作台放松OK"
   TextField "文本域_42" at 395,231 size 57x16; Text '正转条件'
   TextField "文本域_48" at 397,248 size 12x16; Text 'Text'
   IOField "I/O 域_1" at 0,0 size 96x32; FormatPattern 1
      ProcessValue <- "润滑电机工作指示"
   IOField "I/O 域_2" at 0,0 size 96x32; FormatPattern 1
      ProcessValue <- "润滑电机工作指示"
   IOField "I/O 域_3" at 0,0 size 96x32; FormatPattern 1
      ProcessValue <- "润滑电机工作指示"
   IOField "I/O 域_4" at 0,0 size 96x32; FormatPattern 1
      ProcessValue <- "正转条件"
   IOField "I/O 域_5" at 0,0 size 96x32; FormatPattern 1
      ProcessValue <- "主电机启动指示"

screen "润滑状态" 800x480
   IOField "I/O 域_1" at 99,57 size 70x32; FormatPattern 99999
      ProcessValue <- "中间数据.横梁润滑检测时长"
   TextField "文本域_1" at 3,58 size 89x30; Text '横梁润滑检测 时间设定值'
   TextField "文本域_2" at 173,62 size 25x21; Text 'ms'
   IOField "I/O 域_2" at 99,100 size 70x32; FormatPattern 99999
      ProcessValue <- "中间数据.滑块润滑检测时长"
   TextField "文本域_3" at 3,101 size 89x30; Text '滑块润滑检测 时间设定值'
   TextField "文本域_4" at 173,105 size 25x21; Text 'ms'
   IOField "I/O 域_3" at 99,143 size 70x32; FormatPattern 99999
      ProcessValue <- "中间数据.平衡器润滑检测时长"
   TextField "文本域_5" at 3,144 size 89x30; Text '平衡器润滑检 测时间设定值'
   TextField "文本域_6" at 173,148 size 25x21; Text 'ms'
   IOField "I/O 域_4" at 305,61 size 70x32; FormatPattern 99
      ProcessValue <- "中间数据.横梁打油目标次数"
   TextField "文本域_7" at 209,62 size 89x30; Text '横梁润滑检测 次数设定值'
   TextField "文本域_8" at 379,66 size 23x21; Text '次'
   IOField "I/O 域_5" at 305,101 size 70x32; FormatPattern 99
      ProcessValue <- "中间数据.滑块打油目标次数"
   TextField "文本域_9" at 209,102 size 89x30; Text '滑块润滑检测 次数设定值'
   TextField "文本域_10" at 379,106 size 23x21; Text '次'
   IOField "I/O 域_6" at 305,141 size 70x32; FormatPattern 99
      ProcessValue <- "中间数据.平衡器打油目标次数"
   TextField "文本域_11" at 209,142 size 89x30; Text '平衡器润滑检 测次数设定值'
   TextField "文本域_12" at 379,146 size 23x21; Text '次'
   IOField "I/O 域_7" at 474,62 size 53x32; FormatPattern 99
      ProcessValue <- "中间数据.当前打油次数-横梁"
   IOField "I/O 域_9" at 539,64 size 96x32; FormatPattern 99999
      ProcessValue <- "横梁检测当前时间"
   Rectangle "矩形_1" at 27,357 size 96x48
      Appearance <- "辅助中继.横梁润滑故障"
   TextField "文本域_15" at 38,365 size 61x30; Text '横梁 润滑故障'
   Rectangle "矩形_2" at 151,357 size 96x48
      Appearance <- "辅助中继.滑块润滑故障"
   TextField "文本域_16" at 162,365 size 61x30; Text '滑块 润滑故障'
   Rectangle "矩形_3" at 283,357 size 96x48
      Appearance <- "辅助中继.平衡器润滑故障"
   TextField "文本域_17" at 294,365 size 61x30; Text '平衡器 润滑故障'
   Rectangle "矩形_4" at 415,357 size 96x48
      Appearance <- "辅助中继.润滑空开异常"
   TextField "文本域_18" at 429,374 size 61x17; Text '润滑空开'
   Rectangle "矩形_5" at 547,357 size 96x48
      Appearance <- "辅助中继.润滑过滤异常"
   TextField "文本域_19" at 564,374 size 61x17; Text '过滤检测'
   TextField "文本域_14" at 38,219 size 384x31; Text '程序尚未完善， 参数暂勿调整'
   Button "按钮_1" at 17,436 size 94x37; TextOff '滑块角度'
      on Click: ActivateScreen("滑块角度", 0)
   IOField "I/O 域_8" at 474,104 size 53x32; FormatPattern 99
      ProcessValue <- "中间数据.当前打油次数-滑块"
   IOField "I/O 域_10" at 539,106 size 96x32; FormatPattern 99999
      ProcessValue <- "滑块检测当前时间"
   IOField "I/O 域_11" at 474,146 size 53x32; FormatPattern 99
      ProcessValue <- "中间数据.当前打油次数-平衡器"
   IOField "I/O 域_12" at 539,148 size 96x32; FormatPattern 99999
      ProcessValue <- "平衡器检测当前时间"
   TextField "文本域_13" at 477,38 size 61x17; Text '检测次数'
   TextField "文本域_20" at 545,38 size 61x17; Text '当前时间'
*)